(* IEC 61131-3 sources: inproshop/TEAM_V2.0-demo_exported/1.Function/FB/Robot(机械手)/Kuka-四轴, 4 files *)

(* ---- Str_Kuka.st ---- *)
TYPE Str_Kuka :
STRUCT
	Cmd:Str_KukaCmd;//控制
	Status:Str_KukaStatus;//状态
END_STRUCT
END_TYPE

(* ---- Str_KukaCmd.st ---- *)
TYPE Str_KukaCmd :
STRUCT
	Rob_Stop		:BOOL;//停止（Coil 1）
	Rob_Start		:BOOL;//启动（Coil 2）
	Rob_Pause		:BOOL;//暂停（Coil 3）
	Rob_Continue	:BOOL;//继续（Coil 4）
	Rob_Uninatsll	:BOOL;//停止卸载（Coil 5）
	ActiveScara		:BOOL;//激活Scara（Coil 6）
	AppID0			:BOOL;//Main程序编号（Coil 7）
	AppID1			:BOOL;//Main程序编号（Coil 8）
	AppID2			:BOOL;//Main程序编号（Coil 9）
	AppID3			:BOOL;//Main程序编号（Coil 10）
	AppID4			:BOOL;//Main程序编号（Coil 11）
	AppID5			:BOOL;//Main程序编号（Coil 12）
	AppID6			:BOOL;//Main程序编号（Coil 13）
	ShutDown		:BOOL;//重启控制器（Coil 14）
	Acknoledgment	:BOOL;//确认消息（Coil 15）
	MachineIntial	:BOOL;//设备初始化（Coil 16）
	MachineAutoRun	:BOOL;//设备自动中（Coil 17）
	MachineStepRun	:BOOL;//单步信号（Coil 18）
	SpaceBool6		:BOOL;//预备位(Coil 19)
	SpaceBool7		:BOOL;//预备位(Coil 20)
	SpaceBool8		:BOOL;//预备位(Coil 21)
	SpaceBool9		:BOOL;//预备位(Coil 22)
	SpaceBoo20		:BOOL;//预备位(Coil 23)
	SpaceBoo21		:BOOL;//预备位(Coil 24)
	SpaceBoo22		:BOOL;//预备位(Coil 25)
	SpaceBoo23		:BOOL;//预备位(Coil 26)
	SpaceBoo24		:BOOL;//预备位(Coil 27)
	SpaceBoo25		:BOOL;//预备位(Coil 28)
	SpaceBoo26		:BOOL;//预备位(Coil 29)
	SpaceBoo27		:BOOL;//预备位(Coil 30)
	SpaceBoo28		:BOOL;//预备位(Coil 31)
	SpaceBoo29		:BOOL;//预备位(Coil 32)
	InterFace_B		:ARRAY[33..64] OF BOOL;//交互信号
	Speed				:INT;//	运行速度(Holding Register 1)
	ProductType			:INT;//交换数据字(Holding Register 2)
	InterFace_Register3	:INT;//交换数据字(Holding Register 3)
	InterFace_Register4	:INT;//交换数据字(Holding Register 4)
	InterFace_Register5	:INT;//交换数据字(Holding Register 5)
	InterFace_Register6	:INT;//交换数据字(Holding Register 6)
	InterFace_Register7	:INT;//交换数据字(Holding Register 7)
	InterFace_Register8	:INT;//交换数据字(Holding Register 8)
	InterFace_Register9	:INT;//交换数据字(Holding Register 9)
	InterFace_Register10	:INT;//交换数据字(Holding Register 10)
	InterFace_Register11	:INT;//交换数据字(Holding Register 11)
	InterFace_Register12	:INT;//交换数据字(Holding Register 12)
	InterFace_Register13	:INT;//交换数据字(Holding Register 13)
	InterFace_Register14	:INT;//交换数据字(Holding Register 14)
	InterFace_Register15	:INT;//交换数据字(Holding Register 15)
	InterFace_Register16	:INT;//交换数据字(Holding Register 16)

END_STRUCT
END_TYPE

(* ---- Str_KukaStatus.st ---- *)
TYPE Str_KukaStatus :
STRUCT
	Ready:			BOOL;//	系统就绪（Coil 257）
	Running:		BOOL;//	运行中（Coil 258）
	Paused:			BOOL;//	已暂停（Coil 259）
	Stop:			BOOL;//	已停止（Coil 260）
	Error:			BOOL;//	错误-APP（Coil 261）
	SafeguardOn:	BOOL;//	安全门（Coil 262）
	EStopOn:		BOOL;//	急停（Coil 263）
	SError:			BOOL;//	重故障-系统（Coil 264）
	Warning:		BOOL;//	警告（Coil 265）
	Actived:		BOOL;//	已激活（Coil 266）
	ActConfirmed:	BOOL;//	Act已确认（Coil 267）
	Space1:			BOOL;//	预备位（Coil 268）
	Space2:			BOOL;//	预备位（Coil 269）
	Space3:			BOOL;//	预备位（Coil 270）
	Space4:			BOOL;//	预备位（Coil 271）
	Intialed:		BOOL;//	机械手初始化完成（Coil 272）
	InsideBox1:		BOOL;//	Box1（Coil 273）
	InsideBox2:		BOOL;//	Box2（Coil 274）
	InsideBox3:		BOOL;//	Box3（Coil 275）
	InsideBox4:		BOOL;//	Box4（Coil 276）
	InsideBox5:		BOOL;//	Box5（Coil 277）
	InsideBox6:		BOOL;//	Box6（Coil 278）
	InsideBox7:		BOOL;//	Box7（Coil 279）
	InsideBox8:		BOOL;//	Box8 （Coil 280）
	InsideBox9:		BOOL;//	Box9 （Coil 281）
	InsideBox10:	BOOL;//	Box10（Coil 282）
	InsideBox11:	BOOL;//	Box11（Coil 283）
	InsideBox12:	BOOL;//	Box12（Coil 284）
	InsideBox13:	BOOL;//	Box13（Coil 285）
	InsideBox14:	BOOL;//	Box14（Coil 286）
	InsideBox15:	BOOL;//	Box15（Coil 287）
	InsideBox16:	BOOL;//	Box15（Coil 288）
	InsidePlane1:	BOOL;//	Plane1（Coil 289）
	InsidePlane2:	BOOL;//	Plane2（Coil 290）
	InsidePlane3:	BOOL;//	Plane3（Coil 291）
	InsidePlane4:	BOOL;//	Plane4（Coil 292）
	InsidePlane5:	BOOL;//	Plane5（Coil 293）
	InsidePlane6:	BOOL;//	Plane6（Coil 294）
	InsidePlane7:	BOOL;//	Plane7（Coil 295）
	InsidePlane8:	BOOL;//	Plane8（Coil 296）
	InsidePlane9:	BOOL;//	Plane9（Coil 297）
	InsidePlane10:	BOOL;//	Plane10（Coil 298）
	InsidePlane11:	BOOL;//	Plane11（Coil 299）
	InsidePlane12:	BOOL;//	Plane12（Coil 300）
	InsidePlane13:	BOOL;//	Plane13（Coil 301）
	InsidePlane14:	BOOL;// Plane14（Coil 302）
	InsidePlane15:	BOOL;//	Plane15（Coil 303）
	InsidePlane16:	BOOL;//	Plane15（Coil 304）
	InterFace_B:ARRAY[305..336] OF BOOL;//交互信号
	ErrorCode:			WORD;//	错误代码（Holding Register 17）
	InterFace_Register18:	WORD;//	交换数据字(Holding Register18)
	InterFace_Register19:	WORD;// 交换数据字(Holding Register19)
	InterFace_Register20:	WORD;//	交换数据字(Holding Register20)
	InterFace_Register21:	WORD;//	交换数据字(Holding Register21)
	InterFace_Register22:	WORD;//	交换数据字(Holding Register22)
	InterFace_Register23:	WORD;//	交换数据字(Holding Register23)
	InterFace_Register24:	WORD;//	交换数据字(Holding Register24)
	InterFace_Register25:	WORD;//	交换数据字(Holding Register25)
	InterFace_Register26:	WORD;//	交换数据字(Holding Register26)
	InterFace_Register27:	WORD;// 交换数据字(Holding Register27)
	InterFace_Register28:	WORD;//	交换数据字(Holding Register28)
	InterFace_Register29:	WORD;// 交换数据字(Holding Register29)
	InterFace_Register30:	WORD;//	交换数据字(Holding Register30)
	InterFace_Register31:	WORD;//	交换数据字(Holding Register31)
	InterFace_Register32:	WORD;//	交换数据字(Holding Register32)
END_STRUCT
END_TYPE

(* ---- FB_Kuka_V1.st ---- *)
FUNCTION_BLOCK FB_Kuka_V1
VAR_IN_OUT
	ioKuka:Str_Kuka;
END_VAR
VAR_INPUT
	iMode:Str_Mode;//设备控制模式
	iName:WSTRING;//名称
	iDstAdr:STRING;//IP地址
	iDstTcpPort:UINT;//端口号
	iSpeed:REAL;//运行速度
	iProductType:INT;//配方名称
	iClock:BOOL;//发送时钟
END_VAR
VAR_OUTPUT
	oRESET:BOOL;//安全回路复位
	oTimeOut:BOOL;//通讯超时
END_VAR
VAR
	i:INT;//循环变量用
	TcpClient:Str_TcpClient;
	FB_TcpClient_instance:FB_TcpClient;//通讯功能块实例化
	bySendData:ARRAY[0..500]OF BYTE;
	byRevData:ARRAY[0..500]OF BYTE;
	change:INT;//切换读写状态
	TimeDelayExcute:TON;//数据发送间隔
	TimeDelayExcute_R:R_TRIG;
	TimeDelayControl:ARRAY[0..9] OF TON;//控制延时
	TimeOutDelay:TON;//超时
	EnableDelay:TON;//延时使能
END_VAR

ACT_Input();
ACT_Control();
ACT_Output();
ACT_Socket();
